SUBAPPLICATION Uebung_004a11b (* Toggle Flip-Flop mit IE mit BUTTON_SINGLE_CLICK und STORE (NVS) *)
  (* Standard: 61499-2; Description: Copyright (c) 2023 Meisterschulen am Ostbahnhof This program and the accompanying materials are made available under the terms of the Eclipse Public License 2.0 which is available at https://www.eclipse.org/legal/epl-2.0/ SPDX-License-Identifier: EPL-2.0 *)
  (* Version 1.0, 2023-10-23, Franz Höpfinger, Meisterschulen am Ostbahnhof, initial API and implementation and/or initial documentation *)
  PACKAGE Uebungen;
  IMPORT logiBUS::io::DI::logiBUS_DI::Input_I1;
  IMPORT logiBUS::io::DI::logiBUS_DI_Events::BUTTON_SINGLE_CLICK;
  IMPORT logiBUS::io::DQ::logiBUS_DO::Output_Q1;
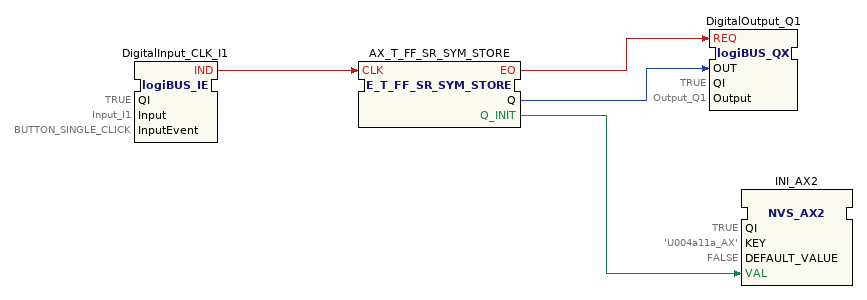
  (* am Anfang letzten Zustand laden! *)
  FBS
    DigitalOutput_Q1 : logiBUS::io::DQ::logiBUS_QX(QI := TRUE, Output := Output_Q1);
    DigitalInput_CLK_I1 : logiBUS::io::DI::logiBUS_IE(QI := TRUE, Input := Input_I1, InputEvent := BUTTON_SINGLE_CLICK);
    AX_T_FF_SR_SYM_STORE : adapter::iec61499::events::E_T_FF_SR_SYM_STORE;
    INI_AX2 : logiBUS::storage::esp32_nvs::NVS_AX2(QI := TRUE, KEY := 'U004a11a_AX', DEFAULT_VALUE := FALSE);
  END_FBS
  EVENT_CONNECTIONS
    DigitalInput_CLK_I1.IND TO AX_T_FF_SR_SYM_STORE.CLK;
    AX_T_FF_SR_SYM_STORE.EO TO DigitalOutput_Q1.REQ;
  END_CONNECTIONS
  DATA_CONNECTIONS
    AX_T_FF_SR_SYM_STORE.Q TO DigitalOutput_Q1.OUT;
  END_CONNECTIONS
  ADAPTER_CONNECTIONS
    AX_T_FF_SR_SYM_STORE.Q_INIT TO INI_AX2.VAL;
  END_CONNECTIONS
END_SUBAPPLICATION
